TYPE "FRK_RegistryRow"
VERSION : 0.1
   STRUCT
      Valid : Bool;
      ModuleType : DInt;
      Parent : Int;
      Exec : DInt;
      ReasonCode : DInt;
      Severity : DInt;
      DataRevision : UDInt;
   END_STRUCT;

END_TYPE
